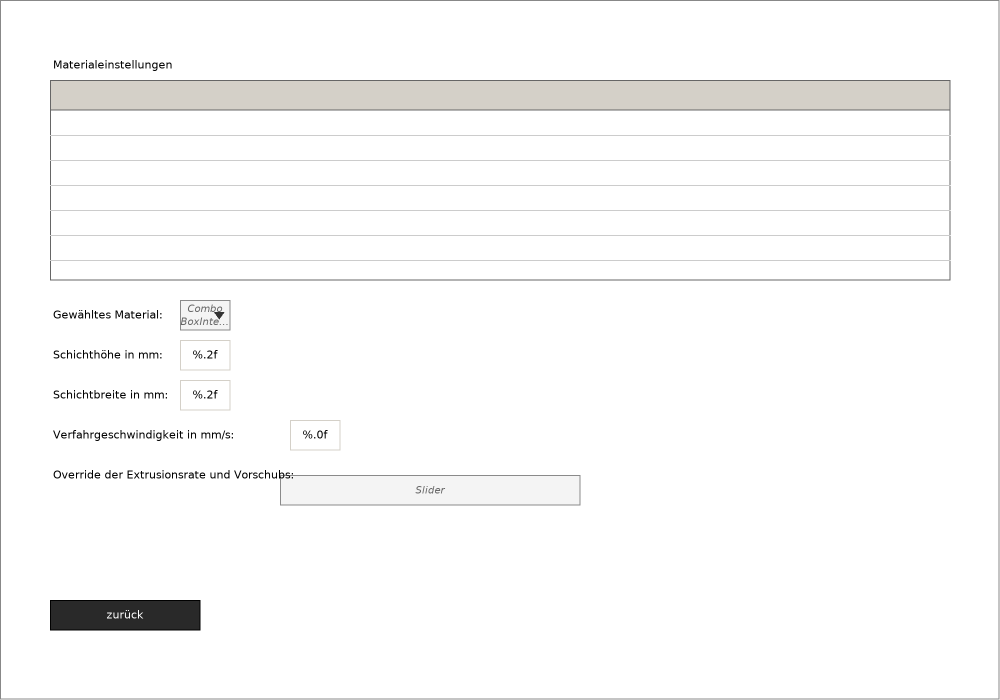
VISUALIZATION V_Konfiguration  // 1000x700
    Table (50,80 900x200), data array: GVL_ParameterExtruder.aMaterialSettings
        p3854506369: GVL_ParameterExtruder.aMaterialSettings[INDEX].sMaterial
        p1892666644: GVL_ParameterExtruder.aMaterialSettings[INDEX].fTempPrintingBed
        p338671338: GVL_ParameterExtruder.aMaterialSettings[INDEX].fTempTop
        p2170511999: GVL_ParameterExtruder.aMaterialSettings[INDEX].fTempMiddle
        p746581629: GVL_ParameterExtruder.aMaterialSettings[INDEX].fFlow2RPM
        p3104783080: GVL_ParameterExtruder.aMaterialSettings[INDEX].fNozzleSizeCoef
        p2232123230: Name
        p511219082: Druckbett Temp.
        p1755163831: Temp. Oben
        p4092479075: Temp. Mitte
        p3723444502: GVL_ParameterExtruder.aMaterialSettings[INDEX].fTempNozzle
        p2237128397: Temp. Düse
        p1218418051: GVL_ParameterExtruder.aMaterialSettings[INDEX].fMaxFlowRate
        p505689113: Max. FlowRate
    Slider (280,475 300x30), variable: GVL_ParameterExtruder.fSpeedOverride, scale 0..100
    ComboBoxInteger (180,300 50x30), variable: GVL_ParameterExtruder.nMaterial
    Label (50,50 150x30), "Materialeinstellungen"
    Label (50,300 150x30), "Gewähltes Material:"
    Label (50,340 150x30), "Schichthöhe in mm:"
    Label (50,380 150x30), "Schichtbreite in mm:"
    Label (50,460 300x30), "Override der Extrusionsrate und Vorschubs:"
    Label (50,420 200x30), "Verfahrgeschwindigkeit in mm/s:"
    Textfield (180,340 50x30), "%.2f", text variable: GVL_ParameterExtruder.fLayerHeight
    Textfield (180,380 50x30), "%.2f", text variable: GVL_ParameterExtruder.fLayerWidth
    Textfield (290,420 50x30), "%.0f", text variable: GVL_ParameterExtruder.fTravelSpeed
    Rectangle (50,600 150x30), "zurück"
        OnMouseDown: change screen: V_Homescreen
END_VISUALIZATION

(* stored: Version 1.1.0.1
   Visu V_Konfiguration: Id {981e287b-265c-4b53-8b9e-caca089d251c} *)
